# B&R Automation Studio project RobotLineDemo (part 4)

### ToolGeo.tool - 5APC4100_TGL4_000/mappMotion/Robots/Gripper/ToolGeo.tool
```
Element RobotTool1_Geometry (Type=tool)
  ToolType = Robot
    Translation:
      Z = -50
```

### ProdLoad1.dynpartable - 5APC4100_TGL4_000/mappMotion/Robots/Product/ProdLoad1.dynpartable
```
Element ProductLoad_1 (Type=dynpartable)
  Row[1]:
    Unit = kg
    Description = Mass
  Row[2]:
    Index = 1
    Unit = m
    Description = Center of gravity - X direction
  Row[3]:
    Index = 2
    Unit = m
    Description = Center of gravity - Y direction
  Row[4]:
    Index = 3
    Unit = m
    Description = Center of gravity - Z direction
  Row[5]:
    Index = 4
    Unit = kg m^2
    Description = Moment of inertia about X
  Row[6]:
    Index = 5
    Unit = kg m^2
    Description = Moment of inertia about Y
  Row[7]:
    Index = 6
    Unit = kg m^2
    Description = Moment of inertia about Z
  Row[8]:
    Index = 1000
    Value = 1
    Unit = 
    Description = 0 (toolDynPar), 1 (productLoadPar)
```

## Logical view

Binary libraries used (declarations not repeated): operator, runtime, AsIecCon, MpBase 6.6.0, McBase 6.9.1, MpAxis 6.9.1, McAcpAx 6.9.1, McPathGen 6.9.1, McAxGroup 6.9.1, McAxis 6.9.1, McProgInt 6.9.1, McTrkPath 6.9.1, MpRobotics 6.9.1

### Global.var - Global variables
```iecst
VAR
	gOverride : REAL;
END_VAR
```


### Program Logical/Tasks/MovePrg (IEC) - Power, Home, Move 

#### Types.typ - Local data types
```iecst
TYPE
	CommandType : 	STRUCT
		Start : BOOL;
		Stop : BOOL;
		ErrorReset : BOOL;
		Settings : CmdSettingsType;
		Details : CmdDetailType;
	END_STRUCT;
	CmdSettingsType : 	STRUCT
		FrameSpaceConveyor1 : LREAL;
		FrameSpaceBetweenTrays : LREAL;
		VelocityConveyor1 : REAL;
		VelocityConveyor2 : REAL;
		HighlightSelectedProducts : BOOL;
	END_STRUCT;
	StateType :
		(
		STARTUP,
		WAIT_FOR_POWER_AND_HOME,
		POWER,
		HOME,
		READ_CURRENT_PARAMETERS,
		START_CONVEYOR_BELTS,
		RUN,
		STOP,
		ERROR_RESET
		);
	GrippedObjectType : 	STRUCT
		OrangeObjectInGripperRob1 : BOOL;
		OrangeObjectInGripperRob2 : BOOL;
		OrangeObjectInGripperRob3 : BOOL;
		OrangeObjectInGripperRob4 : BOOL;
		OrangeObjectInGripperRob5 : BOOL;
		OrangeObjectInGripperRob6 : BOOL;
		GreyObjectInGripperRob1 : BOOL;
		GreyObjectInGripperRob2 : BOOL;
		GreyObjectInGripperRob3 : BOOL;
		GreyObjectInGripperRob4 : BOOL;
		GreyObjectInGripperRob5 : BOOL;
		GreyObjectInGripperRob6 : BOOL;
	END_STRUCT;
	CmdDetailType : 	STRUCT
		MoveConveyor1 : BOOL;
		MoveConveyor2 : BOOL;
		MoveRobotPrograms : BOOL;
		AutoCreationPath1 : BOOL;
		AutoCreationPath2 : BOOL;
		State : StateType;
	END_STRUCT;
END_TYPE
```

#### Variables.var - Local variables
```iecst
(*Command interface*)
VAR
	Cmd : CommandType;
END_VAR
(*Robot and conveyor FBs*)
VAR
	MpRobot_0 : MpDelta4Axis;
	MpRobot_1 : MpDelta4Axis;
	MpRobot_2 : MpDelta4Axis;
	MpRobot_3 : MpDelta4Axis;
	MpRobot_4 : MpDelta4Axis;
	MpRobot_5 : MpDelta4Axis;
	MpRobotPar1 : MpDelta4AxisParType;
	MpRobotPar2 : MpDelta4AxisParType;
	MpRobotPar6 : MpDelta4AxisParType;
	MpAxisConv1 : MpAxisBasic;
	MpAxisConv2 : MpAxisBasic;
	MpAxisParConv1 : MpAxisBasicParType;
	MpAxisParConv2 : MpAxisBasicParType;
	MC_BR_TrackingPathReset_0 : MC_BR_TrackingPathReset;
	MC_BR_TrackingPathReset_1 : MC_BR_TrackingPathReset;
	MC_BR_TrackingFrameDelete_0 : MC_BR_TrackingFrameDelete;
	MC_BR_TrackingFrameDelete_1 : MC_BR_TrackingFrameDelete;
END_VAR
(**)
VAR
	ProcPar_AutCrtCond1TrkPath1_1 : MC_BR_ProcessParam;
	ProcPar_AutCrtCond1TrkPath1_2 : MC_BR_ProcessParam;
	ProcPar_AutCrtCond1TrkPath1_3 : MC_BR_ProcessParam;
	AutoCreateConditionParTrkPath1_1 : McCfgTrkPathAutCrtCondType;
	AutoCreateConditionParTrkPath1_2 : McCfgTrkPathAutCrtCondType;
	AutoCreateConditionParTrkPath1_3 : McCfgTrkPathAutCrtCondType;
	StatusTrackingPath1 : MC_BR_TrackingPathReadStatus;
	StatusTrackingPath2 : MC_BR_TrackingPathReadStatus;
END_VAR
(*Grippers*)
VAR
	GripperRobot1OpenClose : BOOL;
	GripperRobot2OpenClose : BOOL;
	GripperRobot3OpenClose : BOOL;
	GripperRobot4OpenClose : BOOL;
	GripperRobot5OpenClose : BOOL;
	GripperRobot6OpenClose : BOOL;
	GrippersVisu : GrippedObjectType;
END_VAR
(*Create containers*)
VAR
	MC_BR_TrkFrmCreate_Tray : MC_BR_TrackingFrameCreate;
	MC_BR_TrkFrmsCreate_TrayContent : MC_BR_TrackingFramesCreate;
END_VAR
VAR CONSTANT
	NUMBER_OF_FRAMES : USINT := 4;
	NUMBER_OF_FRAMES_INDEX : USINT := NUMBER_OF_FRAMES - 1;
END_VAR
VAR
	TrayContent : ARRAY[0..NUMBER_OF_FRAMES_INDEX] OF McTrkFrmCreateParType;
	MC_BR_TrackingFramesCreate_0 : MC_BR_TrackingFramesCreate;
	i : INT;
	DeltaPos : LREAL;
	TravelAccumulator : LREAL;
	LastConveyorPos : LREAL;
END_VAR
```

### Program Logical/Tasks/Override (IEC)

#### Variables.var - Local variables
```iecst
(*conveyor controller*)
VAR
	Density : REAL; (* items/m*)
	Setpoint : REAL; (* items/m*)
	Slope : REAL; (* % per items/m (e.g., 15.0*)
	MinOverride : REAL;
	MaxOverride : REAL;
	Override : REAL;
	MC_BR_TrackingPathGetFrames_0 : MC_BR_TrackingPathGetFrames;
	frameCount : UINT := 0;
	index : UINT;
	LowerX : LREAL := 0;
	UpperX : LREAL := 0;
	MaxX : LREAL;
	StopZoneReached : BOOL := FALSE;
	McTrkFrmInfoTypeArray : ARRAY[0..499] OF McTrkFrmInfoType;
END_VAR
(*Insert your comment here.*)
VAR
	MC_SetOverride_0 : MC_SetOverride;
END_VAR
```

### pnpPrgR1.st
```iecst
TYPE
	MachineState : (Start, SelectPickPosition, PickObject, SelectPlacePosition, PlaceObject, ParkWithNoObject, ParkWithGrippedObject);
END_TYPE

VAR CONSTANT
	ParkPos      : McPointType := (Pos:=(X:=0, Y:=0, Z:=0));
	PickSynchPosUp   : McPointType := (Pos:=(X:=   0, Y:= 0,  Z:= 70));
	PlaceSynchPosUp   : McPointType := (Pos:=(X:=   0, Y:= 0,  Z:= 70));
    SynchPosDown : McPointType := (Pos:=(X:=   0, Y:= 0,  Z:= 0));
END_VAR

VAR
    TrkFrmID_PickPosition: McTrkFrmIdentType;
    TrkFrmID_PlacePosition: McTrkFrmIdentType;
	State : MachineState;
END_VAR

VAR {AT 'MovePrg'}
	Cmd : CommandType;
END_VAR

PROGRAM _MAIN

    State := MachineState#Start;

    REPEAT
        CASE State OF

        MachineState#Start:
            MoveLR(ParkPos);
            WaitUntilSync(TrackingFrameIsAvailable('ProductSelector'));
            State := MachineState#SelectPickPosition;

        MachineState#SelectPickPosition:
			WaitALAP();
			TrackingFrameSelectorSetAttributeMasks('ProductSelector', 2#0000_0000, 2#0000_0000, 2#0000_0000);
			IF TrackingFrameSelect(TrkFrmID_PickPosition, 'ProductSelector') THEN
				State :=  MachineState#PickObject;
			ELSE
				State := MachineState#ParkWithNoObject;
			END_IF

        MachineState#PickObject:
			IF Cmd.Settings.HighlightSelectedProducts THEN
				TrackingFrameSetAttribute(IP_EVAL(TrkFrmID_PickPosition), 1);
			END_IF
			TrackObjectR(TrkFrmID_PickPosition, PickSynchPosUp, 50, 50);
			MoveLR(SynchPosDown);
			CloseGripper := TRUE;	//close gripper
			WaitTime(0.050);			//wait until gripper is closed [s]
			SetProductLoad('ProductLoad_1');
            MoveLR(PickSynchPosUp);
            State := MachineState#SelectPlacePosition;

        MachineState#SelectPlacePosition:
			WaitALAP();
			TrackingFrameSelectorSetAttributeMasks('PlacePositionSelectorPrior', 2#0000_0001, 2#0000_0000, 2#1100_0000_0000);
            IF TrackingFrameSelect(TrkFrmID_PlacePosition, 'PlacePositionSelectorPrior') THEN
                State :=  MachineState#PlaceObject;
			ELSE
				TrackingFrameSelectorSetAttributeMasks('PlacePositionSelectorPrior', 2#0000_0010, 2#0000_0000, 2#1100_0000_0000);
				IF TrackingFrameSelect(TrkFrmID_PlacePosition, 'PlacePositionSelectorPrior') THEN
					State := MachineState#PlaceObject;
				ELSE

					//Prior area contains no place positions, search in wider area
					TrackingFrameSelectorSetAttributeMasks('PlacePositionSelector', 2#0000_0001, 2#0000_0000, 2#1100_0000_0000);
					IF TrackingFrameSelect(TrkFrmID_PlacePosition, 'PlacePositionSelector') THEN
						State :=  MachineState#PlaceObject;
					ELSE
						TrackingFrameSelectorSetAttributeMasks('PlacePositionSelector', 2#0000_0010, 2#0000_0000, 2#1100_0000_0000);
						IF TrackingFrameSelect(TrkFrmID_PlacePosition, 'PlacePositionSelector') THEN
							State := MachineState#PlaceObject;
						ELSE
							State := MachineState#ParkWithGrippedObject;
						END_IF
					END_IF

				END_IF
			END_IF

        MachineState#PlaceObject:
			TrackObjectR(TrkFrmID_PlacePosition, PlaceSynchPosUp, 50, 50);
			MoveLR(SynchPosDown);
			CloseGripper := FALSE;	//open gripper
			DO_PATH_SYNCH
				TrackingFrameSetAttribute(IP_EVAL(TrkFrmID_PlacePosition), 2048);
			END_PATH_SYNCH
			WaitTime(0.050);		//wait until gripper is opened [s]
			ResetProductLoad();
            MoveLR(PlaceSynchPosUp);
            State := MachineState#SelectPickPosition;

        MachineState#ParkWithNoObject:
			TrackStopR(MachineFrame, ParkPos, 50, 50);
			TrackingFrameSelectorSetAttributeMasks('ProductSelector', 2#0000_0000, 2#0000_0000, 2#0000_0000);
			WaitUntilSync(TrackingFrameSelect(TrkFrmID_PickPosition, 'ProductSelector'));
            State := MachineState#PickObject;

        MachineState#ParkWithGrippedObject:
			TrackStopR(MachineFrame, ParkPos, 50, 50);

			TrackingFrameSelectorSetAttributeMasks('PlacePositionSelector', 2#0000_0000, 2#0000_0000, 2#1100_0000_0000);
			WaitUntilSync(TrackingFrameIsAvailable('PlacePositionSelector'));

			TrackingFrameSelectorSetAttributeMasks('PlacePositionSelectorPrior', 2#0000_0001, 2#0000_0000, 2#1100_0000_0000);
			IF TrackingFrameSelect(TrkFrmID_PlacePosition, 'PlacePositionSelectorPrior') THEN
				State :=  MachineState#PlaceObject;
			ELSE
				TrackingFrameSelectorSetAttributeMasks('PlacePositionSelectorPrior', 2#0000_0010, 2#0000_0000, 2#1100_0000_0000);
				IF TrackingFrameSelect(TrkFrmID_PlacePosition, 'PlacePositionSelectorPrior') THEN
					State := MachineState#PlaceObject;
				ELSE

					//Prior area contains no place positions, search in wider area
					TrackingFrameSelectorSetAttributeMasks('PlacePositionSelector', 2#0000_0001, 2#0000_0000, 2#1100_0000_0000);
					IF TrackingFrameSelect(TrkFrmID_PlacePosition, 'PlacePositionSelector') THEN
						State :=  MachineState#PlaceObject;
					ELSE
						TrackingFrameSelectorSetAttributeMasks('PlacePositionSelector', 2#0000_0010, 2#0000_0000, 2#1100_0000_0000);
						IF TrackingFrameSelect(TrkFrmID_PlacePosition, 'PlacePositionSelector') THEN
							State := MachineState#PlaceObject;
						ELSE
							State := MachineState#ParkWithGrippedObject;
						END_IF
					END_IF

				END_IF
			END_IF

		END_CASE

	UNTIL FALSE END_REPEAT;

END_PROGRAM
```

### pnpPrgR2.st
```iecst
TYPE
	MachineState : (Start, SelectPickPosition, PickObject, SelectPlacePosition, PlaceObject, ParkWithNoObject, ParkWithGrippedObject);
END_TYPE

VAR CONSTANT
    ParkPos      : McPointType := (Pos:=(X:=0, Y:=0, Z:=0));
	PickSynchPosUp   : McPointType := (Pos:=(X:=   0, Y:= 0,  Z:= 70));
	PlaceSynchPosUp   : McPointType := (Pos:=(X:=   0, Y:= 0,  Z:= 70));
    SynchPosDown : McPointType := (Pos:=(X:=   0, Y:= 0,  Z:= 0));
END_VAR

VAR
    TrkFrmID_PickPosition: McTrkFrmIdentType;
    TrkFrmID_PlacePosition: McTrkFrmIdentType;
	State : MachineState;
END_VAR

VAR {AT 'MovePrg'}
	Cmd : CommandType;
END_VAR

PROGRAM _MAIN

    State := MachineState#Start;

    REPEAT
        CASE State OF

        MachineState#Start:
            MoveLR(ParkPos);
            WaitUntilSync(TrackingFrameIsAvailable('ProductSelector'));
            State := MachineState#SelectPickPosition;

        MachineState#SelectPickPosition:
			WaitALAP();
			TrackingFrameSelectorSetAttributeMasks('ProductSelector', 2#0000_0000, 2#0000_0000, 2#0000_0000);
			IF TrackingFrameSelect(TrkFrmID_PickPosition, 'ProductSelector') THEN
				State :=  MachineState#PickObject;
			ELSE
				State := MachineState#ParkWithNoObject;
			END_IF

		MachineState#PickObject:
			IF Cmd.Settings.HighlightSelectedProducts THEN
				TrackingFrameSetAttribute(IP_EVAL(TrkFrmID_PickPosition), 1);
			END_IF
            TrackObjectR(TrkFrmID_PickPosition, PickSynchPosUp, 50, 50);
			MoveLR(SynchPosDown);
				CloseGripper := TRUE;	//close gripper
			WaitTime(0.050);			//wait until gripper is closed [s]
			SetProductLoad('ProductLoad_1');
            MoveLR(PickSynchPosUp);
            State := MachineState#SelectPlacePosition;

        MachineState#SelectPlacePosition:
			WaitALAP();
			TrackingFrameSelectorSetAttributeMasks('PlacePositionSelector', 2#0000_0001, 2#0000_0000, 2#1100_0000_0000);
            IF TrackingFrameSelect(TrkFrmID_PlacePosition, 'PlacePositionSelector') THEN
                State :=  MachineState#PlaceObject;
			ELSE
				TrackingFrameSelectorSetAttributeMasks('PlacePositionSelector', 2#0000_0010, 2#0000_0000, 2#1100_0000_0000);
				IF TrackingFrameSelect(TrkFrmID_PlacePosition, 'PlacePositionSelector') THEN
					State := MachineState#PlaceObject;
				ELSE
					State := MachineState#ParkWithGrippedObject;
				END_IF
			END_IF

        MachineState#PlaceObject:
            TrackObjectR(TrkFrmID_PlacePosition, PlaceSynchPosUp, 50, 50);
			MoveLR(SynchPosDown);
			CloseGripper := FALSE;	//open gripper
			DO_PATH_SYNCH
				TrackingFrameSetAttribute(IP_EVAL(TrkFrmID_PlacePosition), 2048);
			END_PATH_SYNCH
			WaitTime(0.050);		//wait until gripper is opened [s]
			ResetProductLoad();
            MoveLR(PlaceSynchPosUp);
            State := MachineState#SelectPickPosition;

        MachineState#ParkWithNoObject:
			TrackStopR(MachineFrame, ParkPos, 50, 50);
			TrackingFrameSelectorSetAttributeMasks('ProductSelector', 2#0000_0000, 2#0000_0000, 2#0000_0000);
			WaitUntilSync(TrackingFrameSelect(TrkFrmID_PickPosition, 'ProductSelector'));
            State := MachineState#PickObject;

        MachineState#ParkWithGrippedObject:
			TrackStopR(MachineFrame, ParkPos, 50, 50);

			TrackingFrameSelectorSetAttributeMasks('PlacePositionSelector', 2#0000_0000, 2#0000_0000, 2#1100_0000_0000);
			WaitUntilSync(TrackingFrameIsAvailable('PlacePositionSelector'));

			TrackingFrameSelectorSetAttributeMasks('PlacePositionSelector', 2#0000_0001, 2#0000_0000, 2#1100_0000_0000);
			IF TrackingFrameSelect(TrkFrmID_PlacePosition, 'PlacePositionSelector') THEN
				State :=  MachineState#PlaceObject;
			ELSE
				TrackingFrameSelectorSetAttributeMasks('PlacePositionSelector', 2#0000_0010, 2#0000_0000, 2#1100_0000_0000);
				IF TrackingFrameSelect(TrkFrmID_PlacePosition, 'PlacePositionSelector') THEN
					State := MachineState#PlaceObject;
				ELSE
					State := MachineState#ParkWithGrippedObject;
				END_IF
			END_IF

		END_CASE

	UNTIL FALSE END_REPEAT;

END_PROGRAM
```

- Product.tnr (not shown)

- Tray.tnr (not shown)

- tray 100x100.tnr (not shown)

- donut.tnr (not shown)

- tray 300x200.tnr (not shown)

- Middle_Belt.tnr (not shown)

- Leg_Belt.tnr (not shown)

- Leg.tnr (not shown)

- Front_Belt.tnr (not shown)

- Front.tnr (not shown)

- Back.tnr (not shown)

- Back_Belt.tnr (not shown)

- Middle.tnr (not shown)

- Product.tnr (not shown)

- Tray.tnr (not shown)

- tray 100x100.tnr (not shown)

- donut.tnr (not shown)

- tray 300x200.tnr (not shown)

- Middle_Belt.tnr (not shown)

- Leg_Belt.tnr (not shown)

- Leg.tnr (not shown)

- Front_Belt.tnr (not shown)

- Front.tnr (not shown)

- Back.tnr (not shown)

- Back_Belt.tnr (not shown)

- Middle.tnr (not shown)

Listed in the project but not available here: Logical/Tasks/MovePrg/Main.st, Logical/Tasks/MovePrg/Action.st, Logical/Tasks/Override/Main.st, Logical/Tasks/Override/Actions.st, Logical/UserPartitionData/MotionPrg/pnpPrgR6.st
